// TwinCAT 3 PLC project PLC
// ProgramVersion: 3.1.4023.0
// libraries:
//   Tc2_Standard, * (Beckhoff Automation GmbH)
//   Tc2_System, * (Beckhoff Automation GmbH)
//   Tc3_Module, * (Beckhoff Automation GmbH)
// project tree:
//   DUTs/ ST_TrafficLight.TcDUT
//   / PlcTask.TcTTO
//   POUs/ FB_TrafficLightHandler.TcPOU, MAIN.TcPOU
// real-time tasks:
//   TASK PlcTask: cycle T#10ms, priority 20, ADS port 350

CONFIGURATION PLC
    RESOURCE PLC ON TwinCAT3
        TASK PlcTask(INTERVAL := T#10ms, PRIORITY := 20);
        PROGRAM MAIN WITH PlcTask : MAIN;
    END_RESOURCE
END_CONFIGURATION

// ---- DUTs/ST_TrafficLight.TcDUT
TYPE ST_TrafficLight :
STRUCT
	
RedLight 	: BOOL := FALSE;
YellowLight : BOOL := FALSE;
GreenLight 	: BOOL := FALSE;


END_STRUCT
END_TYPE

// ---- POUs/MAIN.TcPOU
PROGRAM MAIN
VAR
	
// Users can read pragmas in TcHmi
trafficLight01 	: ST_TrafficLight;

// These are user defined pragams which can bring meaning to different symbol instances
{attribute 'Access' := 'Admin'}
trafficLight02 	: ST_TrafficLight;

{attribute 'Theme' := 'Dark'}
trafficLight03 	: ST_TrafficLight;

TrafficLightHandler : FB_TrafficLightHandler;


NonTrafficLightSymbol : BOOL;

END_VAR

END_PROGRAM

// ---- POUs/FB_TrafficLightHandler.TcPOU
FUNCTION_BLOCK FB_TrafficLightHandler
VAR_INPUT
END_VAR
VAR_OUTPUT
END_VAR
VAR
	
Lights : ST_TrafficLight;

END_VAR

{attribute 'TcRpcEnable'}
METHOD M_RequestAllLightOff : BOOL
VAR_INPUT
END_VAR
Lights.GreenLight :=FALSE;
Lights.YellowLight := FALSE;
Lights.RedLight := FALSE;
END_METHOD

{attribute 'TcRpcEnable'}
METHOD M_RequestAllLightOn : BOOL
VAR_INPUT
END_VAR
Lights.GreenLight := TRUE;
Lights.YellowLight := TRUE;
Lights.RedLight := TRUE;
END_METHOD

END_FUNCTION_BLOCK
